TYPE "udt_FlyingCarriage_Config"
VERSION : 0.1
// Block: udt_FlyingCarriage_Config
   STRUCT
      SLS_VEL : LReal;
      DelayMissingCondition : Time;
      Fan : Struct
         Exist : Bool;
         DelayOff : Time;
      END_STRUCT;
   END_STRUCT;

END_TYPE
